// TIA Portal V20 export
DATA_BLOCK "Alarms"   // DB8
{ DB_Accessible_From_OPC_UA := 'FALSE' }
AUTHOR : ERsystem_FA2_DH. Kim
// stored: Access Published, DBAccessibleFromOPCUA false, DBAccessibleFromWebserver false, MemoryReserve 100, Namespace Unit1
   VAR
      unitAlarms { ExternalWritable := 'False'} : "LAF_typeAlarms";
      emAlarms { ExternalWritable := 'False'} : Array[0.._.U1_NO_OF_EMs] of "LAF_typeAlarms";
      maintenanceFaults { ExternalWritable := 'False'} : Array[0..199] of Bool;   // PFE Maintenance Faults
      productionFaults { ExternalWritable := 'False'} : Array[0..199] of Bool;   // PFE Production Faults
      toolingFault { ExternalWritable := 'False'} : Array[0..199] of Bool;   // PFE Tooling Faults
      qualityFault { ExternalWritable := 'False'} : Array[0..199] of Bool;   // PFE Quality Faults
      throughputFaultBlocked { ExternalWritable := 'False'} : Array[0..199] of Bool;   // PFE Throughput Fault Blocked
      throughputFaultStarved { ExternalWritable := 'False'} : Array[0..199] of Bool;   // PFE Throughput Fault Starved
      throughputFault { ExternalWritable := 'False'} : Array[0..199] of Bool;   // PFE Throughput Fault
      systemFaultGeneral { ExternalWritable := 'False'} : Array[0..199] of Bool;   // PFE System Fault General
      materialFault { ExternalWritable := 'False'} : Array[0..199] of Bool;   // PFE Material Fault
      maintenanceWarnings { ExternalWritable := 'False'} : Array[0..199] of Bool;   // PFE Maintenance Warnings
      productionWarning { ExternalWritable := 'False'} : Array[0..199] of Bool;   // PFE Production Warning
      toolingWarning { ExternalWritable := 'False'} : Array[0..199] of Bool;   // PFE Tooling Warning
      qualityWarning { ExternalWritable := 'False'} : Array[0..199] of Bool;   // PFE Quality Warning
      throughputWarning { ExternalWritable := 'False'} : Array[0..199] of Bool;   // PFE Throughput Warning
      systemWarning { ExternalWritable := 'False'} : Array[0..199] of Bool;   // PFE System Warning
      materialWarning { ExternalWritable := 'False'} : Array[0..199] of Bool;   // PFE Material Warning
      maintenanceStatus { ExternalWritable := 'False'} : Array[0..199] of Bool;   // PFE Maintenance Status
      productionStatus { ExternalWritable := 'False'} : Array[0..199] of Bool;   // PFE Production Status
      toolingStatus { ExternalWritable := 'False'} : Array[0..199] of Bool;   // PFE Tooling Status
      qualityStatus { ExternalWritable := 'False'} : Array[0..199] of Bool;   // PFE Quality Status
      throughputStatus { ExternalWritable := 'False'} : Array[0..199] of Bool;   // PFE Throughput Status
      systemStatus { ExternalWritable := 'False'} : Array[0..199] of Bool;   // PFE System Status
      materialStatus { ExternalWritable := 'False'} : Array[0..199] of Bool;   // PFE Material Status
      tonMaintenanceFault { ExternalWritable := 'False'} : Array[0..199] of TON_TIME;   // PFE Maintenance Faults Ton Timer
      tonProductionFault { ExternalWritable := 'False'} : Array[0..199] of TON_TIME;   // PFE Production Faults Ton Timer
      tonToolingFault { ExternalWritable := 'False'} : Array[0..199] of TON_TIME;   // PFE Tooling Faults Ton Timer
      tonQualityFault { ExternalWritable := 'False'} : Array[0..199] of TON_TIME;   // PFE Quality Faults Ton Timer
      tonThroughputFaultBlocked { ExternalWritable := 'False'} : Array[0..199] of TON_TIME;   // PFE Throughput Fault Blocked Ton Timer
      tonThroughputFaultStarved { ExternalWritable := 'False'} : Array[0..199] of TON_TIME;   // PFE Throughput Fault Starved Ton Timer
      tonThroughputFault { ExternalWritable := 'False'} : Array[0..199] of TON_TIME;   // PFE Throughput Fault Ton Timer
      tonSystemFaultGeneral { ExternalWritable := 'False'} : Array[0..199] of TON_TIME;   // PFE System Fault General Ton Timer
      tonMaterialFault { ExternalWritable := 'False'} : Array[0..199] of TON_TIME;   // PFE Material Fault Ton Timer
      tonMaintenanceWarning { ExternalWritable := 'False'} : Array[0..199] of TON_TIME;   // PFE Maintenance Warnings Ton Timer
      tonProductionWarning { ExternalWritable := 'False'} : Array[0..199] of TON_TIME;   // PFE Production Warning Ton Timer
      tonToolingWarning { ExternalWritable := 'False'} : Array[0..199] of TON_TIME;   // PFE Tooling Warning Ton Timer
      tonQualityWarning { ExternalWritable := 'False'} : Array[0..199] of TON_TIME;   // PFE Quality Warning Ton Timer
      tonThroughputWarning { ExternalWritable := 'False'} : Array[0..199] of TON_TIME;   // PFE Throughput Warning Ton Timer
      tonSystemWarning { ExternalWritable := 'False'} : Array[0..199] of TON_TIME;   // PFE System Warning Ton Timer
      tonMaterialWarning { ExternalWritable := 'False'} : Array[0..199] of TON_TIME;   // PFE Material Warning Ton Timer
      tonMaintenanceStatus { ExternalWritable := 'False'} : Array[0..199] of TON_TIME;   // PFE Maintenance Status Ton Timer
      tonProductionStatus { ExternalWritable := 'False'} : Array[0..199] of TON_TIME;   // PFE Production Status Ton Timer
      tonToolingStatus { ExternalWritable := 'False'} : Array[0..199] of TON_TIME;   // PFE Tooling Status Ton Timer
      tonQualityStatus { ExternalWritable := 'False'} : Array[0..199] of TON_TIME;   // PFE Quality Status Ton Timer
      tonThroughputStatus { ExternalWritable := 'False'} : Array[0..199] of TON_TIME;   // PFE Throughput Status Ton Timer
      tonSystemStatus { ExternalWritable := 'False'} : Array[0..199] of TON_TIME;   // PFE System Status Ton Timer
      tonMaterialStatus { ExternalWritable := 'False'} : Array[0..199] of TON_TIME;   // PFE Material Status Ton Timer
      TonTimer { ExternalWritable := 'False'} : Array[0..99] of TON_TIME;
   END_VAR
BEGIN
   // maintenanceFaults[0] : EM Error
   // maintenanceFaults[10] : Brake time test after 24Hours Faults
   // maintenanceFaults[20] : CV Cover All Not OK Faults
   // systemFaultGeneral[0] : MOTOR POWER MCFEEDBACK
   // systemFaultGeneral[1] : E202CB_MOTOR POWER TRIPPED
   // systemFaultGeneral[2] : E208CB_MAIN CONTROL PANELMAIN POWER TRIPPED
   // systemFaultGeneral[3] : E320CB_E9304PWS CONTROLPOWER SMPS AC POWERTRIPPED
   // systemFaultGeneral[4] : E326CB_E9404PWS CONTROLPOWER SMPS AC POWERTRIPPED
   // systemFaultGeneral[5] : E400CB_COMPENSATOR X-AXISPOWER TR PRIMARYTRIPPED
   // systemFaultGeneral[6] : E410CB_COMPENSATOR X-AXISPOWER TR ECONDARYTRIPPED
   // systemFaultGeneral[7] : E500CB_SEPA P&P X-AXIS POWERTR PRIMARY TRIPPED
   // systemFaultGeneral[8] : E510CB_SEPA P&P X-AXIS POWERTR ECONDARY TRIPPED
   // systemFaultGeneral[9] : E720CB_POWER METER POWERTRIIPED
   // systemFaultGeneral[10] : E726CB_POWER METER CONTROLPOWER TRIIPED
   // systemFaultGeneral[11] : E3304CB_COMPENSATOR X-AXISPOWER ON TRIPPRED
   // systemFaultGeneral[12] : E3504CB_SPEA P&P 1 X-AXISPOWER ON TRIPPED
   // systemFaultGeneral[13] : E3604CB_SPEA P&P 2 X-AXISPOWER ON TRIPPED
   // systemFaultGeneral[14] : E7116CB_PROCESSOR POWER ONTRIPPRED
   // systemFaultGeneral[15] : E7156CB_MAIN CONTROL PANELHOT POWER TRIPPED
   // systemFaultGeneral[16] : E7304CB_PANEL LED POWERTRIPPED
   // systemFaultGeneral[17] : E8100CB_120VAC CONTROL POWERTR PRIMARY TRIPPED
   // systemFaultGeneral[18] : E8110CB_120VAC CONTROL POWERTR SECONDARY TRIPPED
   // systemFaultGeneral[19] : E8116CB_CONTROL POWER ONTRIPPED
   // systemFaultGeneral[20] : E8156CB_MAIN CONTROL PANELCONTROL POWERTRIPPED
   // systemFaultGeneral[21] : E9104PWS_CONTROL POWER SMPSDC OK
   // systemFaultGeneral[22] : E9122CB_ENCODER, TERMINALUNIT CONTROL POWERTRIPPED
   // systemFaultGeneral[23] : E9128CB_SERVO CONTROL UNITCONTROL POWERTRIPPED
   // systemFaultGeneral[24] : E9204CB_PANEL FAN POWERTRIPPED
   // systemFaultGeneral[25] : E9304PWS_CONTROL POWER SMPSDC OK
   // systemFaultGeneral[26] : E9306CB_CONTROL DC POWERTRIPPED
   // systemFaultGeneral[27] : E9316CB_SERVO CONTROL POWERTRIPPED
   // systemFaultGeneral[28] : E9404PWS_CONTROL POWER SMPSDC OK
   // systemFaultGeneral[29] : E9406CB_CONTROL DC POWERTRIPPED
   // systemFaultGeneral[30] : E9416CB_JUNCTION BOX CLASS 2SMPS TRIPPED
   // systemFaultGeneral[31] : E9422CB_EQUIPMENT LED POWERTRIPPED
   // systemFaultGeneral[32] : E214CB_E6404PWS CONTROLLER POWER SMPS AC POWER TRIPPED
   // systemFaultGeneral[33] : E222CB_E6704PWS CONTROLLER POWER SMPS AC POWER TRIPPED
   // systemFaultGeneral[34] : E226CB_E6804PWS SAFETY POWER SMPS AC POWER TRIPPED
   // systemFaultGeneral[35] : E4120CB_PROCESSOR POWER ON TIPPRED
   // systemFaultGeneral[36] : E4126CB_PROGRAMING POWER OUTLET TRPPED
   // systemFaultGeneral[37] : E4304CB_PANEL LED POWER TRIPPED
   // systemFaultGeneral[38] : E4420CB_CONTROL LEVEL HUB POWER TRIPPED
   // systemFaultGeneral[39] : E4426CB_MAIN HMI POWER TRIPPED
   // systemFaultGeneral[40] : E4432CB_PORTABLE HMI POWER TIPPED
   // systemFaultGeneral[41] : E4604CB_PANEL IRT HUB POWER TIPPED
   // systemFaultGeneral[42] : E4608ES_IRT HUB FAULT
   // systemFaultGeneral[43] : E5110CB_120VAC CONTROL POWER TR SECONDARY TRIPPED
   // systemFaultGeneral[44] : E5120CB_CONTROL POWER ON TRIPPED
   // systemFaultGeneral[45] : E5126CB_VISION MONITOR-1&MCU POWER STRIP OUTLET POWER TRIPPED
   // systemFaultGeneral[46] : E5132CB_VISION MONITOR-2&VISION MONITOR-3 POWER STRIP OUTLET POWER TRIPPED
   // systemFaultGeneral[47] : E5156CB_VISION LIGHT CONTROLLER POWER STRIP OUTLET POWER TRIPPED
   // systemFaultGeneral[48] : E5222CB_FFU POWER-1 POWER TRIPPED
   // systemFaultGeneral[49] : E6154CB_ET200MP I/O OUTPUT POWER TRIPPED
   // systemFaultGeneral[50] : E6180CB_JUNCTION BOX CONTROL POWER TRIPPED
   // systemFaultGeneral[51] : E6204CB_CLASS 2 SMPS POWER TRIPPED
   // systemFaultGeneral[52] : E6220CB_ET200ECO PN-1 POWER TRIPPED
   // systemFaultGeneral[53] : E6224CB_ET200ECO PN-2 POWER TRIPPED
   // systemFaultGeneral[54] : E6228CB_ET200ECO PN-3 POWER TRIPPED
   // systemFaultGeneral[55] : E6232CB_ET200ECO PN-4 POWER TRIPPED
   // systemFaultGeneral[56] : E6304CB_PANEL FAN POWER TRIPPED
   // systemFaultGeneral[57] : E6406CB_CONTROLLER DC POWER TRIPPED
   // systemFaultGeneral[58] : E6422CB_MANIFOLD-1 CONTROL POWER TRIPPED
   // systemFaultGeneral[59] : E6430CB_MANIFOLD-2 CONTROL POWER TRIPPED
   // systemFaultGeneral[60] : E6456CB_DRIVE-CLIQ HUB POWER TRIPPED
   // systemFaultGeneral[61] : E6462CB_DRIVE-CLIQ HUB POWER TRIPPED
   // systemFaultGeneral[62] : E6468CB_HANDY QR READER POWER TRIPPED
   // systemFaultGeneral[63] : E6474CB_VISION CONTROLLER-1 POWER TRIPPED
   // systemFaultGeneral[64] : E6480CB_VISION CONTROLLER-2 POWER TRIPPED
   // systemFaultGeneral[65] : E6486CB_VISION CONTROLLER-3 POWER TRIPPED
   // systemFaultGeneral[66] : E6506CB_LINE LASER MODULE-1 POWER TRIPPED
   // systemFaultGeneral[67] : E6512CB_LINE LASER MODULE-2 POWER TRIPPED
   // systemFaultGeneral[68] : E6706CB_CONTROLLER DC POWER TRIPPED
   // systemFaultGeneral[69] : E6716CB_EPC CONTROLLER-1 POWER TRIPPED
   // systemFaultGeneral[70] : E6722CB_EPC CONTROLLER-2 POWER TRIPPED
   // systemFaultGeneral[71] : E6728CB_EPC CONTROLLER-3 POWER TRIPPED
   // systemFaultGeneral[72] : E6734CB_EPC CONTROLLER-4 POWER TRIPPED
   // systemFaultGeneral[73] : E6806CB_SAFETY DC POWER TRIPPED
   // systemFaultGeneral[74] : E6816CB_ET200SP I/O SAFETY POWER TRIPPED
   // systemFaultGeneral[75] : E6836CB_JUNCTION BOX CONTROL POWER TRIPPED
   // systemFaultGeneral[76] : E6856CB_ET200ECO PN SAFETYT-1 POWER TRIPPED
   // systemFaultGeneral[77] : E6862CB_ET200ECO PN SAFETYT-2 POWER TRIPPED
   // systemFaultGeneral[78] : E6756CB_DC-DC CONVERTER IN POWER TRIPPED
   // systemFaultGeneral[79] : E6762CB_HOT WIRE CUTTER POWER TRIPPED
   // systemFaultGeneral[80] : E110CB_MAIN HMI POWER TRIPPED
   // systemFaultGeneral[81] : E4404PWS_PLC POWER SMPS DC NG
   // systemFaultGeneral[82] : E6104PWS_CONTROL POWER SMPS DC NG
   // systemFaultGeneral[83] : E6206PWS_CLASS 2 SMPS MONITORING NG
   // systemFaultGeneral[84] : E6404PWS_CONTROLLER POWER SMPS DC NG
   // systemFaultGeneral[85] : E6704PWS_CONTROLLER POWER SMPS DC NG
   // systemFaultGeneral[86] : E6804PWS_SAFETY POWER SMPS DC NG
   // systemFaultGeneral[115] : Main Pressure Switch-1 Fault
   // systemFaultGeneral[116] : Main Pressure Switch-2 Fault
   // maintenanceWarnings[10] : 8 Hours Time Over
   // maintenanceWarnings[20] : Cathode Conveyor Cover Open
   // maintenanceWarnings[21] : Anode Conveyor Cover Open
   // maintenanceWarnings[22] : BA60 External Door Open
   // maintenanceWarnings[25] : BA10 SCS Mode Select
   // maintenanceWarnings[26] : BA15 SCS Mode Select
   // maintenanceWarnings[27] : BA30 SCS Mode Select
   // maintenanceWarnings[28] : BA60 SCS Mode Select
   // maintenanceWarnings[30] : Brake test not ready warning
END_DATA_BLOCK
